Fanuc KAREL source: ks00040.KL

-- PROVISIONAL review KL for V1013-1; original PC SHA256 c8a14e741d05f64af652b63a8ff9d90529c7d88241c9157a62b8f974c9079ceb
-- Incomplete behavior may be omitted. Consult companion uncertainty JSON. Do not deploy.
PROGRAM KS00040
%NOLOCKGROUP
BEGIN
  -- UNRESOLVED_PC offsets 5-13; opcodes 3F,75
  -- UNRESOLVED_PC offsets 18-27; opcodes 3F,75
  -- UNRESOLVED_PC offsets 32-45; opcodes 22,1D,23
  -- UNRESOLVED_PC offsets 50-54; opcodes 7F
END KS00040
